(* Logix 5000 project; controller cal1615 1756-L62 rev 20.11; software revision 20.05; part 50 of 82 *)
(* tags used below, declared in another part *)
   FAULT : BOOL;   // Fault AFI
   metering_roll_alarm : TIMER;
   metering_roll_close : TIMER;
   p01_recipe_active : recipe;   // Active Recipe
   p01r02 : routine;   // System Misc Control
   p01r09_pb_global_reset : BOOL;   // System Modes PB: Global Fault Reset
   p02_dint_from_hmi : hmi_dint;
   p11r02_shutdown_temp : BOOL;   // Zone 1 Misc Control Safe Shutdown Temperature
   p11r30 : routine;   // Zone 1 Temperature Control
   p12r02_shutdown_temp : BOOL;   // Zone 2 Misc Control Safe Shutdown Temperature
   p12r30 : routine;   // Zone 2 Temperature Control
   p23_ai_ds_gap_dint : DINT;
   p23_ai_ds_masked_gap : REAL;
   p23_ai_lfl : REAL;   // Impreg Inputs LFL level
   p23_ai_metering_roll_amps : REAL;   // Impreg Analog Input Impreg Metering Roll Motor Current
   p23_ai_metering_roll_hz : REAL;   // Impreg Analog Input Impreg Metering Roll Motor Max Hz
   p23_ai_metering_roll_speed_fpm : REAL;   // Impreg Analog Input Impreg Roll Speed
   p23_ai_prs : REAL;   // Impreg Analog Inputs Impreg Enclosure Pressure
   p23_ai_servo_ds_position : REAL;   // Impreg Servo Drive Side Actual Position
   p23_ai_servo_ds_torque : REAL;   // Impreg Servo Drive Side Actual Torque
   p23_ai_servo_ds_velocity : REAL;   // Impreg Servo Drive Side Velocity Feedback
   p23_ai_servo_os_position : REAL;   // Impreg Inputs Servo Operator Side Position
   p23_ai_servo_os_velocity : REAL;   // Impreg Inputs Servo Operator Side Velocity
   p23_ai_supply_amps : REAL;   // Impreg Analog Inputs Supply Fan VFD Amps
   p23_ai_supply_hz : REAL;   // Impreg Analog Inputs Supply Fan VFD Hz
   p23_ai_supply_rpm : REAL;   // Impreg Analog Inputs Supply Fan RPM
   p23_ctr_gear_ratio : REAL;
   p23_ctr_lfl_input_max : REAL;
   p23_ctr_lfl_input_min : REAL;
   p23_ctr_lfl_output_max : REAL;
   p23_ctr_lfl_output_min : REAL;
   p23_ctr_roll_diameter_ft : REAL;
   p23_di_exhaust_speed_ok : BOOL;
   p23_di_filter_clean : BOOL;
   p23_di_impreg_exhaust_running : BOOL;
   p23_di_impreg_tank_up : BOOL;   // Input Impreg Dip Tank Up
   p23_di_metering_bar_close : BOOL;   // Impreg Input SSS: Metering Bar Close
   p23_di_metering_bar_open : BOOL;   // Impreg Input SSS: Metering Bar Open
   p23_di_metering_roll : acs800_di_normal;   // Impreg Digital Inputs Metering Roll VFD
   p23_di_servo_ds : servo_di;   // Impreg Digital Inputs Servo Drive Side
   p23_di_servo_os : servo_di;   // Impreg Digital Inputs Servo Operator Side
   p23_di_splice_jump : BOOL;   // Impreg Inputs PB: Splice Jump
   p23_di_spring : acs800_di_normal;
   p23_di_srv_ds_ok : BOOL;   // Impreg Inputs Metering Servo Drive Side Ok
   p23_di_srv_op_ok : BOOL;   // Impreg Inputs Metering Servo Operator Side Ok
   p23_di_supply : acs800_di_normal;   // Impreg Supply VFD VFD Inputs
   p23_di_supply_motor_therm : BOOL;   // Impreg Inputs Supply Fan Motor Thermostat
   p23_di_supply_speed_ok : BOOL;
   p23_di_tank_level_high : BOOL;   // Impreg Input Dip Impreg Level High
   p23_di_tank_level_low : BOOL;   // Impreg Input Dip Impreg Level Low
   p23_di_therm : BOOL;   // Impreg Inputs Metering Roll Motor Temperature Ok
   p23_di_though_level_low : BOOL;   // Impreg Input Dip Impreg Through Level Low
   p23_di_vfd_jog_fwd : BOOL;   // Impreg Input PB: VFD Jog FWD
   p23_di_vfd_jog_rev : BOOL;   // Impreg Input PB: VFD Jog REV
   p23_dint_to_hmi : DINT[17];   // Impreg Dint to HMI
   p23_do_enable_impreg_exhaust_fan : BOOL;   // Impreg Enclosure Digital Output Exhaust Fan Enable
   p23_do_impreg_nip_close : BOOL;   // Impreg Digital Output Impreg Nip close
   p23_param_lfl_hhl : REAL;   // Impreg Parameter LFL High High Limit
   p23_param_lfl_hl : REAL;   // Impreg Parameters LFL High Limit
   p23_param_servo_open_position : REAL;
   p23_param_zone_pressure : REAL;   // MOP HMI Iface Parameters Minimum Pressure
   p23r01 : routine;   // Impreg Main
   p23r02 : routine;   // Impreg Misc Control
   p23r02_fault_exists : BOOL;
   p23r02_open_pos_dint : DINT;
   p23r02_open_pos_real : REAL;
   p23r02_pb_start_exh : BOOL;
   p23r02_pb_stop_exh : BOOL;
   p23r02_request_nip_close : BOOL;   // Impreg Misc Control Request Nip Close
   p23r02_timer_fault : TIMER[4];   // Impreg Misc Control Timer Fault
   p23r02_timer_warning : TIMER[4];   // Impreg Misc Control Timer Warning
   p23r02_unack_fault : BOOL;   // Imperg Misc Control Unackn. Fault Exist
   p23r02_unack_warning : BOOL;   // Impreg Misc Control Unackn. Warning Exist
   p23r02_warning_exists : BOOL;
   p23r03 : routine;   // Impreg Inputs
   p23r03_hz : SYS_SCP;   // Impreg Roll Analog Inputs SCP Hz
   p23r03_impreg_lfl_monitor : SYS_SCP;   // Impreg Analog Inputs LFL Monitor Scaling
   p23r03_impreg_prs_input_max : REAL;
   p23r03_impreg_prs_input_min : REAL;
   p23r03_impreg_prs_output_max : REAL;
   p23r03_impreg_prs_output_min : REAL;
   p23r03_impreg_prs_scp : SYS_SCP;   // Impreg Analog Input Impreg Enclosure Pressure
   p23r03_metering_vfd_rpm_to_speed : SYS_RPM_TO_SPEED;   // Impreg Metering Roll Input VFD AI
   p23r04 : routine;   // Impreg Outputs
   p23r05 : routine;   // Impreg Dint to HMI
   p23r06 : routine;   // Impreg Real to HMI
   p23r07 : routine;   // Impreg Alarms
   p23r08 : routine;   // Impreg Warnings
   p23r09 : routine;   // Impreg Mode Selection
   p23r11 : routine;   // Impreg Servo Operator Side
   p23r12 : routine;   // Impreg Servo Drive Side
   p23r15 : routine;   // Impreg Metering Roll VFD
   p23r17_di_brake : BOOL;
   p23r17_di_therm : BOOL;

PROGRAM P23_Impreg   (* main routine R01_Main *)
VAR
   jog : BOOL;
   metering_roll : TIMER := (PRE := 4500);
   p23r17 : routine := (comment := -1073741714, fault := 48, fault_ack := 48);
   p23r17_request_line_run : BOOL;
END_VAR

ROUTINE R01_Main   (* ladder *)
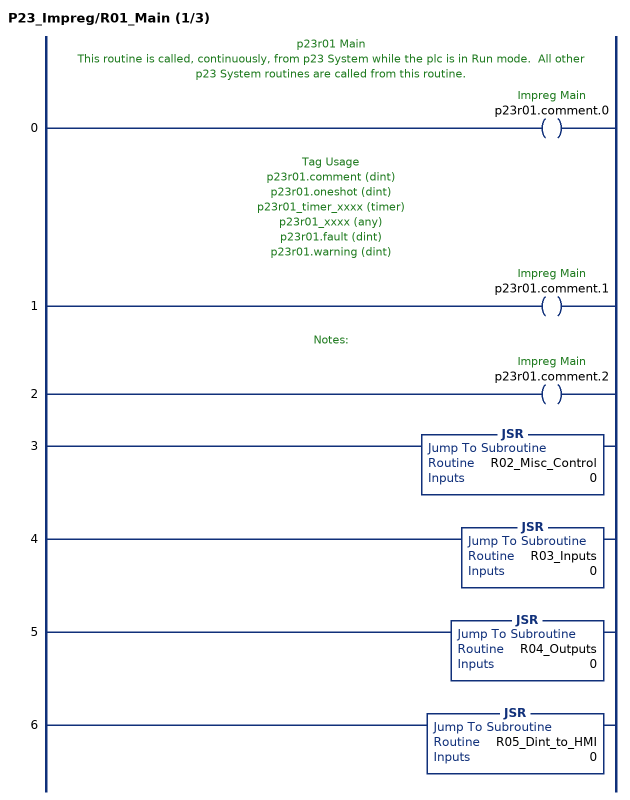
   // p23r01 Main
   // This routine is called, continuously, from p23 System while the plc is in Run mode.  All other p23 System routines are called from this routine.
   0: OTE(p23r01.comment.0);
   // Tag Usage
   // p23r01.comment (dint)
   // p23r01.oneshot (dint)
   // p23r01_timer_xxxx (timer)
   // p23r01_xxxx (any)
   // p23r01.fault (dint)
   // p23r01.warning (dint)
   1: OTE(p23r01.comment.1);
   // Notes:
   2: OTE(p23r01.comment.2);
   3: JSR(R02_Misc_Control,0);
   4: JSR(R03_Inputs,0);
   5: JSR(R04_Outputs,0);
   6: JSR(R05_Dint_to_HMI,0);
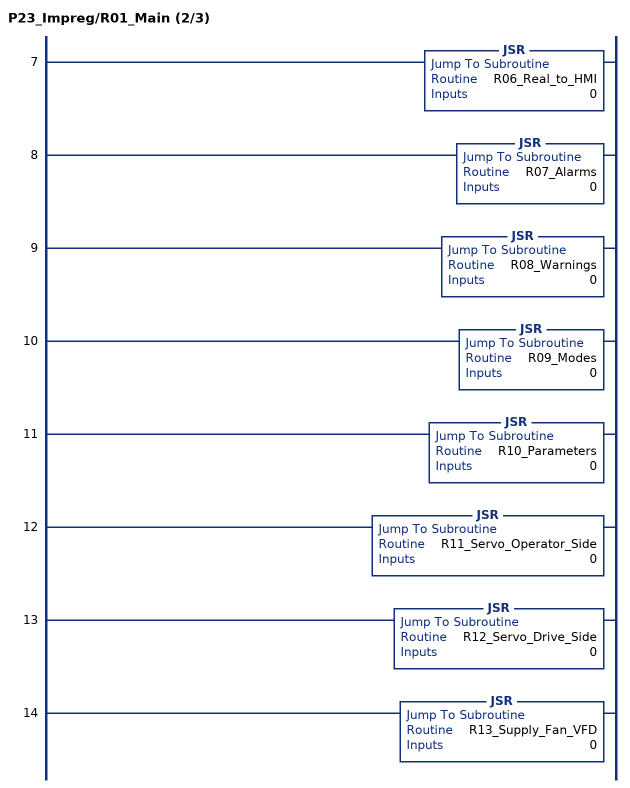
   7: JSR(R06_Real_to_HMI,0);
   8: JSR(R07_Alarms,0);
   9: JSR(R08_Warnings,0);
   10: JSR(R09_Modes,0);
   11: JSR(R10_Parameters,0);
   12: JSR(R11_Servo_Operator_Side,0);
   13: JSR(R12_Servo_Drive_Side,0);
   14: JSR(R13_Supply_Fan_VFD,0);
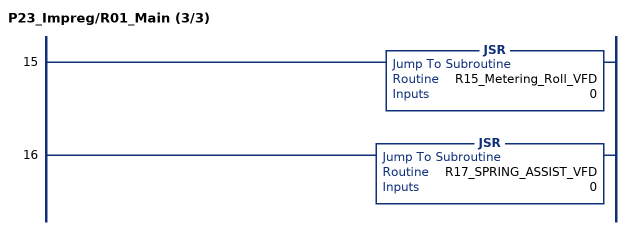
   15: JSR(R15_Metering_Roll_VFD,0);
   16: JSR(R17_SPRING_ASSIST_VFD,0);
END_ROUTINE

ROUTINE R02_Misc_Control   (* ladder *)
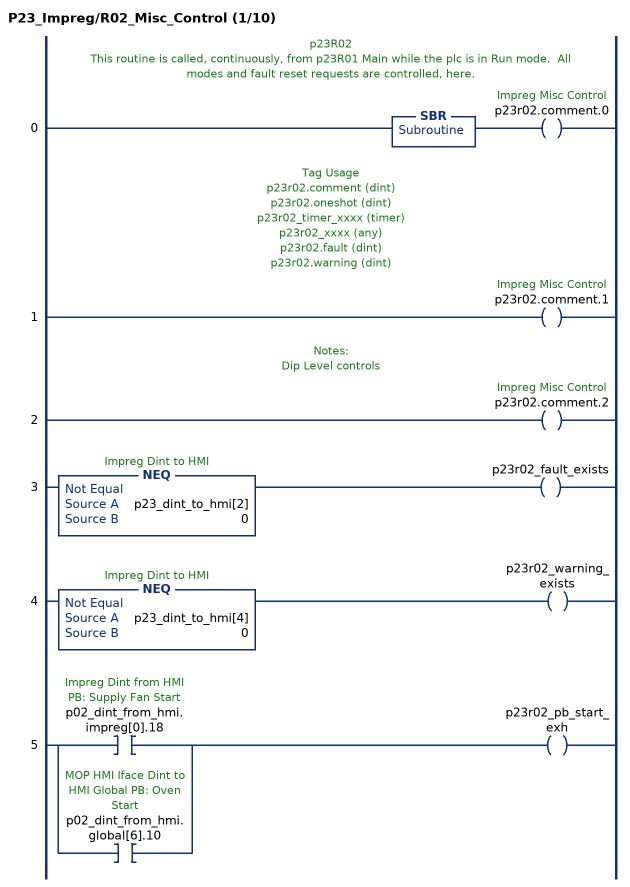
   // p23R02
   // This routine is called, continuously, from p23R01 Main while the plc is in Run mode.  All modes and fault reset requests are controlled, here.
   0: SBR()OTE(p23r02.comment.0);
   // Tag Usage
   // p23r02.comment (dint)
   // p23r02.oneshot (dint)
   // p23r02_timer_xxxx (timer)
   // p23r02_xxxx (any)
   // p23r02.fault (dint)
   // p23r02.warning (dint)
   1: OTE(p23r02.comment.1);
   // Notes:
   // Dip Level controls
   2: OTE(p23r02.comment.2);
   3: NEQ(p23_dint_to_hmi[2],0)OTE(p23r02_fault_exists);
   4: NEQ(p23_dint_to_hmi[4],0)OTE(p23r02_warning_exists);
   5: [XIC(p02_dint_from_hmi.impreg[0].18) ,XIC(p02_dint_from_hmi.global[6].10) ]OTE(p23r02_pb_start_exh);
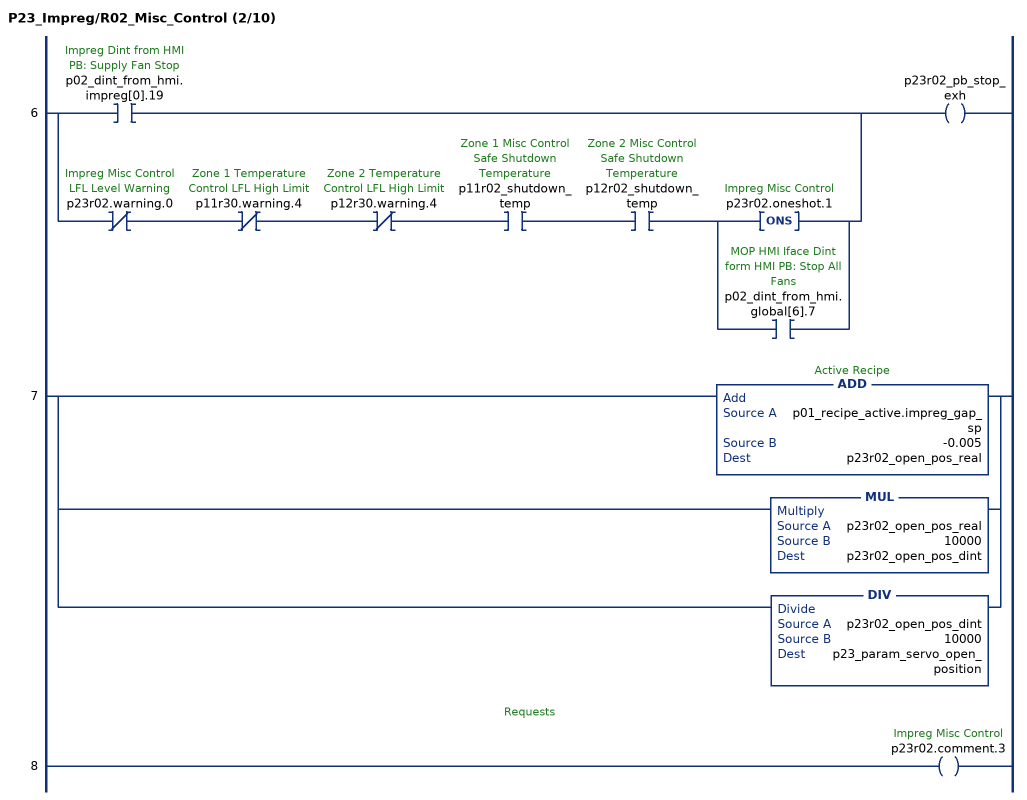
   6: [XIC(p02_dint_from_hmi.impreg[0].19) ,XIO(p23r02.warning.0) XIO(p11r30.warning.4) XIO(p12r30.warning.4) XIC(p11r02_shutdown_temp) XIC(p12r02_shutdown_temp) [ONS(p23r02.oneshot.1) ,XIC(p02_dint_from_hmi.global[6].7) ] ]OTE(p23r02_pb_stop_exh);
   7: [ADD(p01_recipe_active.impreg_gap_sp,-0.005,p23r02_open_pos_real) ,MUL(p23r02_open_pos_real,10000,p23r02_open_pos_dint) ,DIV(p23r02_open_pos_dint,10000,p23_param_servo_open_position) ];
   // Requests
   8: OTE(p23r02.comment.3);
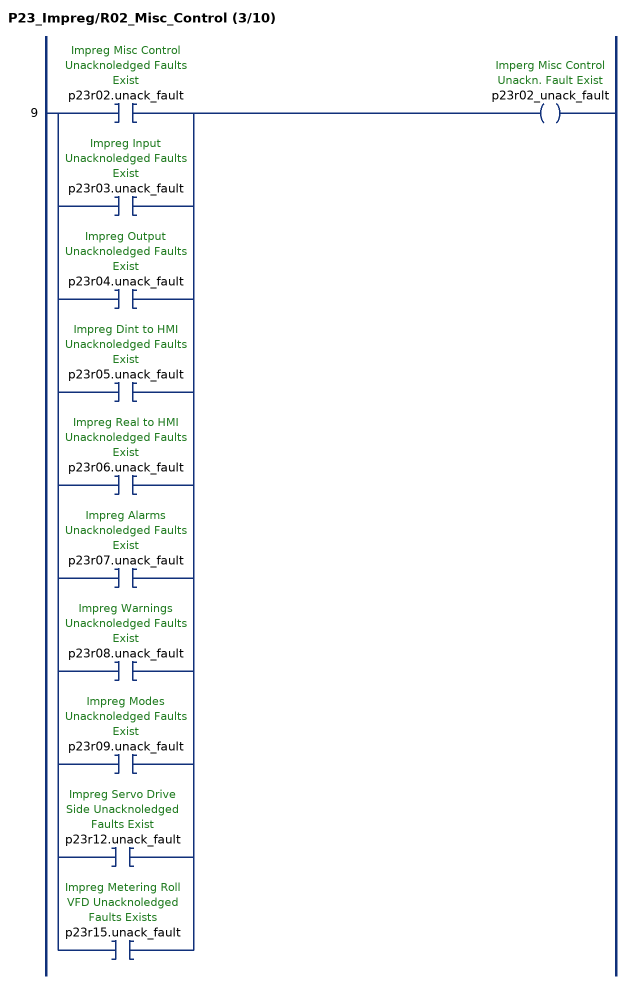
   9: [XIC(p23r02.unack_fault) ,XIC(p23r03.unack_fault) ,XIC(p23r04.unack_fault) ,XIC(p23r05.unack_fault) ,XIC(p23r06.unack_fault) ,XIC(p23r07.unack_fault) ,XIC(p23r08.unack_fault) ,XIC(p23r09.unack_fault) ,XIC(p23r12.unack_fault) ,XIC(p23r15.unack_fault) ]OTE(p23r02_unack_fault);
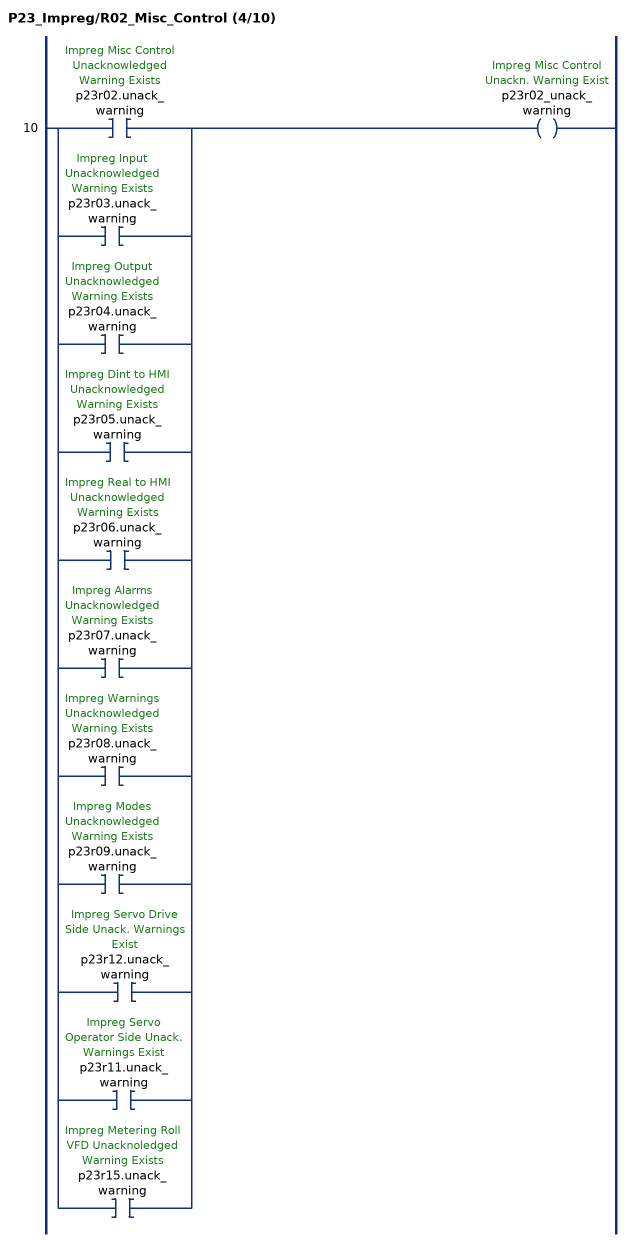
   10: [XIC(p23r02.unack_warning) ,XIC(p23r03.unack_warning) ,XIC(p23r04.unack_warning) ,XIC(p23r05.unack_warning) ,XIC(p23r06.unack_warning) ,XIC(p23r07.unack_warning) ,XIC(p23r08.unack_warning) ,XIC(p23r09.unack_warning) ,XIC(p23r12.unack_warning) ,XIC(p23r11.unack_warning) ,XIC(p23r15.unack_warning) ]OTE(p23r02_unack_warning);
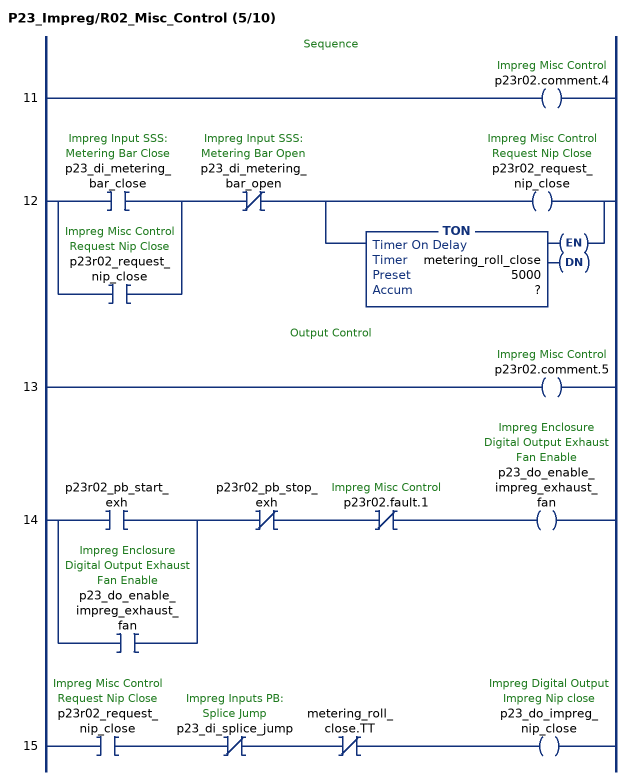
   // Sequence
   11: OTE(p23r02.comment.4);
   12: [XIC(p23_di_metering_bar_close) ,XIC(p23r02_request_nip_close) ]XIO(p23_di_metering_bar_open)[OTE(p23r02_request_nip_close) ,TON(metering_roll_close,?,?) ];
   // Output Control
   13: OTE(p23r02.comment.5);
   14: [XIC(p23r02_pb_start_exh) ,XIC(p23_do_enable_impreg_exhaust_fan) ]XIO(p23r02_pb_stop_exh)XIO(p23r02.fault.1)OTE(p23_do_enable_impreg_exhaust_fan);
   15: XIC(p23r02_request_nip_close)XIO(p23_di_splice_jump)XIO(metering_roll_close.TT)OTE(p23_do_impreg_nip_close);
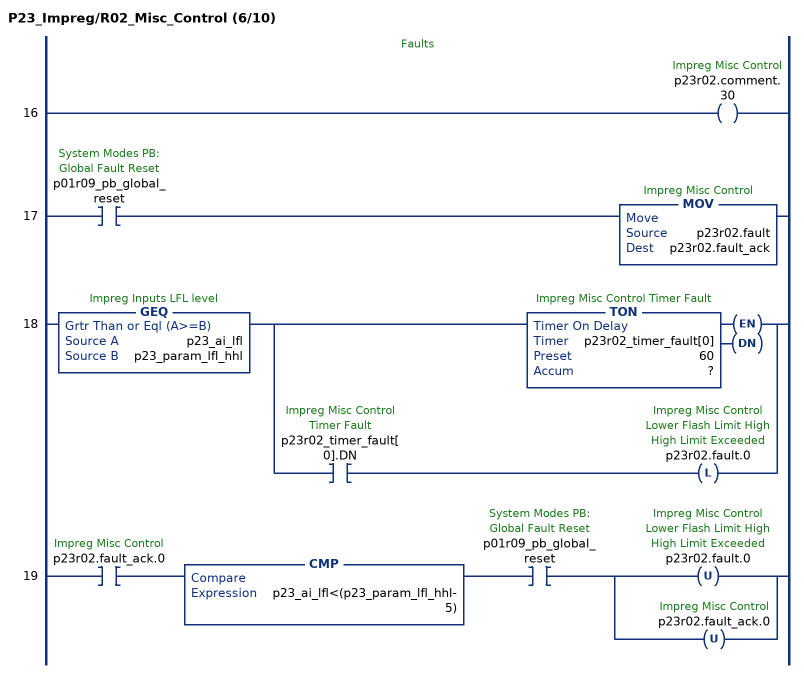
   // Faults
   16: OTE(p23r02.comment.30);
   17: XIC(p01r09_pb_global_reset)MOV(p23r02.fault,p23r02.fault_ack);
   18: GEQ(p23_ai_lfl,p23_param_lfl_hhl)[TON(p23r02_timer_fault[0],?,?) ,XIC(p23r02_timer_fault[0].DN) OTL(p23r02.fault.0) ];
   19: XIC(p23r02.fault_ack.0)CMP(p23_ai_lfl<(p23_param_lfl_hhl-5))XIC(p01r09_pb_global_reset)[OTU(p23r02.fault.0) ,OTU(p23r02.fault_ack.0) ];
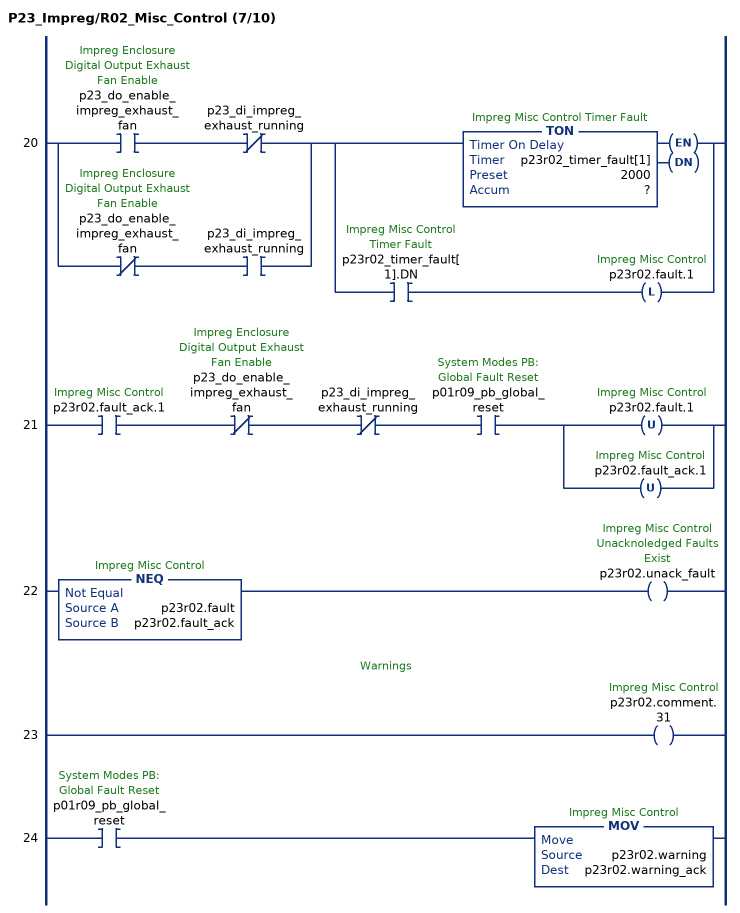
   20: [XIC(p23_do_enable_impreg_exhaust_fan) XIO(p23_di_impreg_exhaust_running) ,XIO(p23_do_enable_impreg_exhaust_fan) XIC(p23_di_impreg_exhaust_running) ][TON(p23r02_timer_fault[1],?,?) ,XIC(p23r02_timer_fault[1].DN) OTL(p23r02.fault.1) ];
   21: XIC(p23r02.fault_ack.1)XIO(p23_do_enable_impreg_exhaust_fan)XIO(p23_di_impreg_exhaust_running)XIC(p01r09_pb_global_reset)[OTU(p23r02.fault.1) ,OTU(p23r02.fault_ack.1) ];
   22: NEQ(p23r02.fault,p23r02.fault_ack)OTE(p23r02.unack_fault);
   // Warnings
   23: OTE(p23r02.comment.31);
   24: XIC(p01r09_pb_global_reset)MOV(p23r02.warning,p23r02.warning_ack);
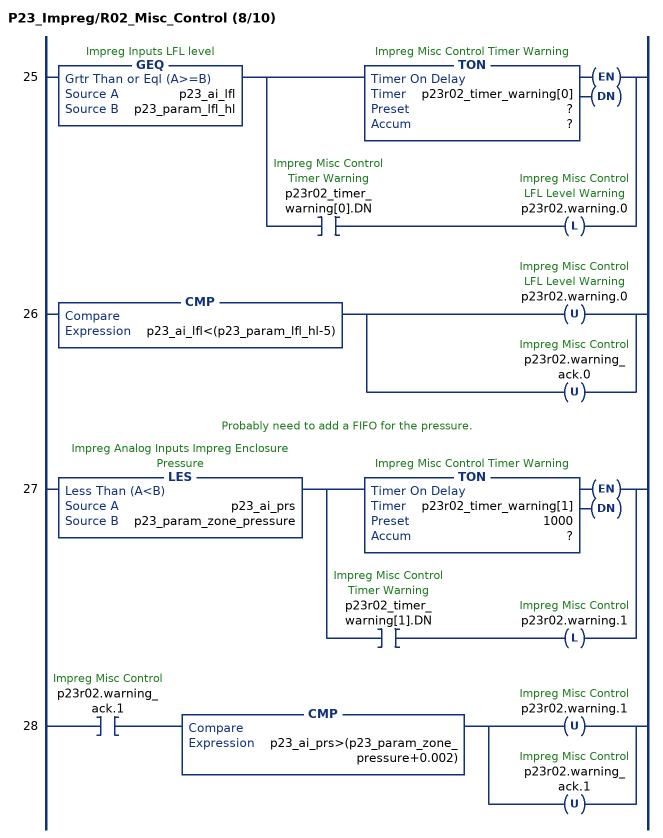
   25: GEQ(p23_ai_lfl,p23_param_lfl_hl)[TON(p23r02_timer_warning[0],?,?) ,XIC(p23r02_timer_warning[0].DN) OTL(p23r02.warning.0) ];
   26: CMP(p23_ai_lfl<(p23_param_lfl_hl-5))[OTU(p23r02.warning.0) ,OTU(p23r02.warning_ack.0) ];
   // Probably need to add a FIFO for the pressure.
   27: LES(p23_ai_prs,p23_param_zone_pressure)[TON(p23r02_timer_warning[1],?,?) ,XIC(p23r02_timer_warning[1].DN) OTL(p23r02.warning.1) ];
   28: XIC(p23r02.warning_ack.1)CMP(p23_ai_prs>(p23_param_zone_pressure+0.002))[OTU(p23r02.warning.1) ,OTU(p23r02.warning_ack.1) ];
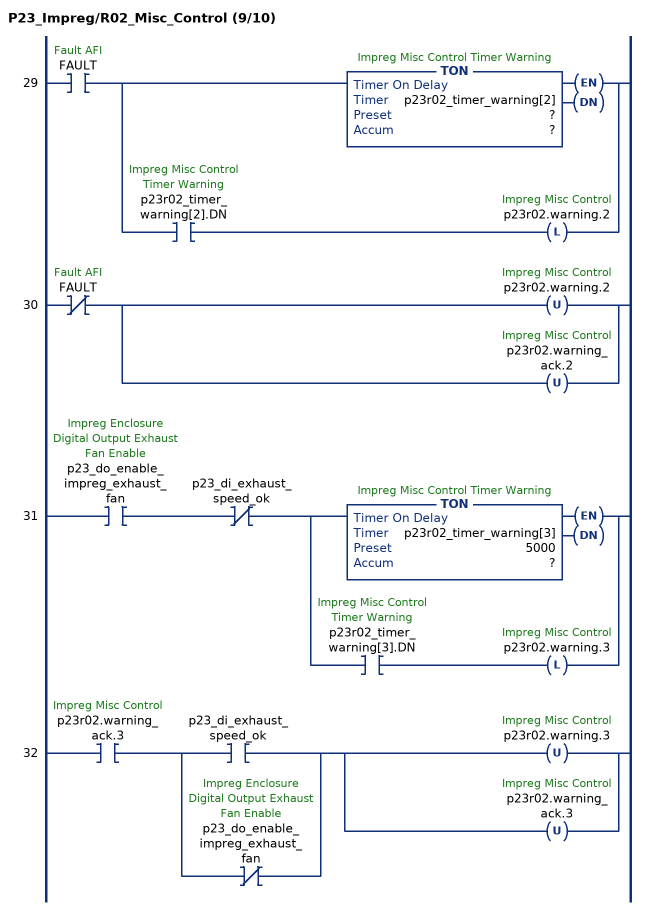
   29: XIC(FAULT)[TON(p23r02_timer_warning[2],?,?) ,XIC(p23r02_timer_warning[2].DN) OTL(p23r02.warning.2) ];
   30: XIO(FAULT)[OTU(p23r02.warning.2) ,OTU(p23r02.warning_ack.2) ];
   31: XIC(p23_do_enable_impreg_exhaust_fan)XIO(p23_di_exhaust_speed_ok)[TON(p23r02_timer_warning[3],?,?) ,XIC(p23r02_timer_warning[3].DN) OTL(p23r02.warning.3) ];
   32: XIC(p23r02.warning_ack.3)[XIC(p23_di_exhaust_speed_ok) ,XIO(p23_do_enable_impreg_exhaust_fan) ][OTU(p23r02.warning.3) ,OTU(p23r02.warning_ack.3) ];
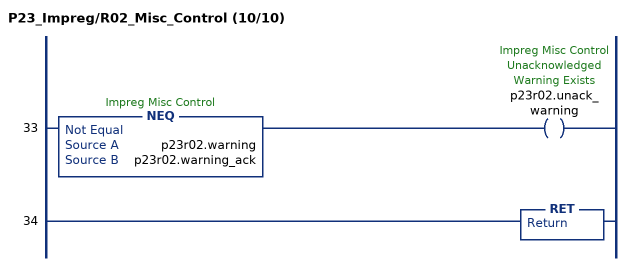
   33: NEQ(p23r02.warning,p23r02.warning_ack)OTE(p23r02.unack_warning);
   34: RET();
END_ROUTINE

ROUTINE R03_Inputs   (* ladder *)
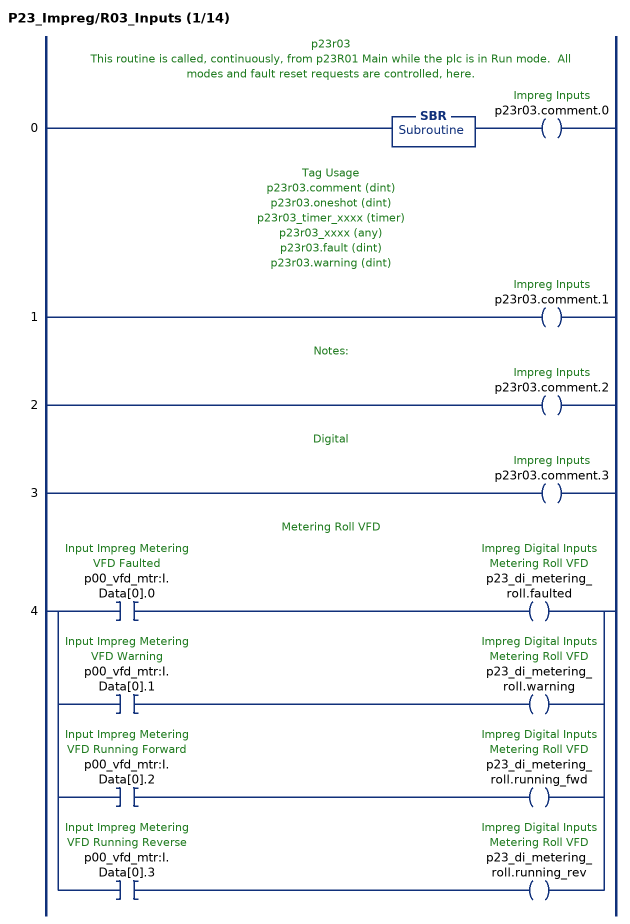
   // p23r03
   // This routine is called, continuously, from p23R01 Main while the plc is in Run mode.  All modes and fault reset requests are controlled, here.
   0: SBR()OTE(p23r03.comment.0);
   // Tag Usage
   // p23r03.comment (dint)
   // p23r03.oneshot (dint)
   // p23r03_timer_xxxx (timer)
   // p23r03_xxxx (any)
   // p23r03.fault (dint)
   // p23r03.warning (dint)
   1: OTE(p23r03.comment.1);
   // Notes:
   2: OTE(p23r03.comment.2);
   // Digital
   3: OTE(p23r03.comment.3);
   // Metering Roll VFD
   4: [XIC(p00_vfd_mtr:I.Data[0].0) OTE(p23_di_metering_roll.faulted) ,XIC(p00_vfd_mtr:I.Data[0].1) OTE(p23_di_metering_roll.warning) ,XIC(p00_vfd_mtr:I.Data[0].2) OTE(p23_di_metering_roll.running_fwd) ,XIC(p00_vfd_mtr:I.Data[0].3) OTE(p23_di_metering_roll.running_rev) ];
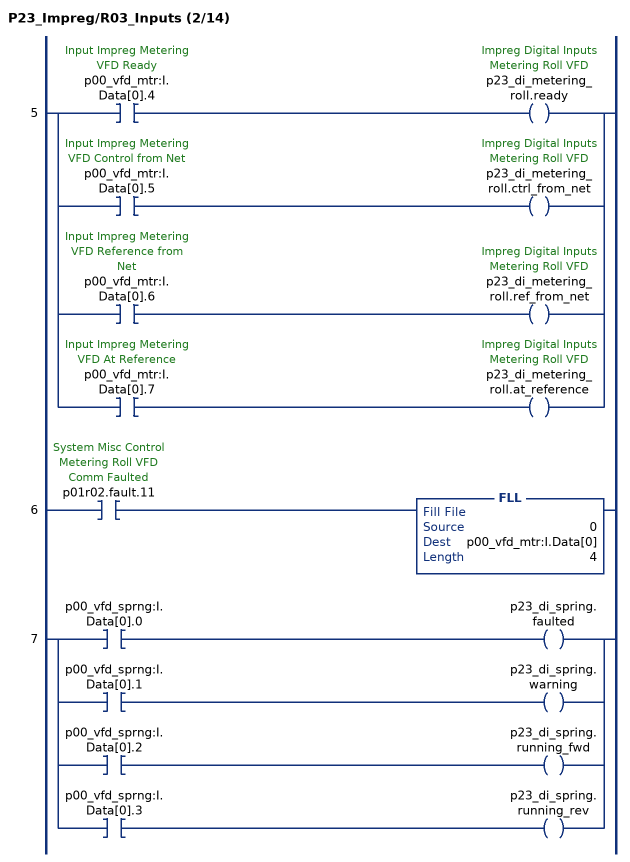
   5: [XIC(p00_vfd_mtr:I.Data[0].4) OTE(p23_di_metering_roll.ready) ,XIC(p00_vfd_mtr:I.Data[0].5) OTE(p23_di_metering_roll.ctrl_from_net) ,XIC(p00_vfd_mtr:I.Data[0].6) OTE(p23_di_metering_roll.ref_from_net) ,XIC(p00_vfd_mtr:I.Data[0].7) OTE(p23_di_metering_roll.at_reference) ];
   6: XIC(p01r02.fault.11)FLL(0,p00_vfd_mtr:I.Data[0],4);
   7: [XIC(p00_vfd_sprng:I.Data[0].0) OTE(p23_di_spring.faulted) ,XIC(p00_vfd_sprng:I.Data[0].1) OTE(p23_di_spring.warning) ,XIC(p00_vfd_sprng:I.Data[0].2) OTE(p23_di_spring.running_fwd) ,XIC(p00_vfd_sprng:I.Data[0].3) OTE(p23_di_spring.running_rev) ];
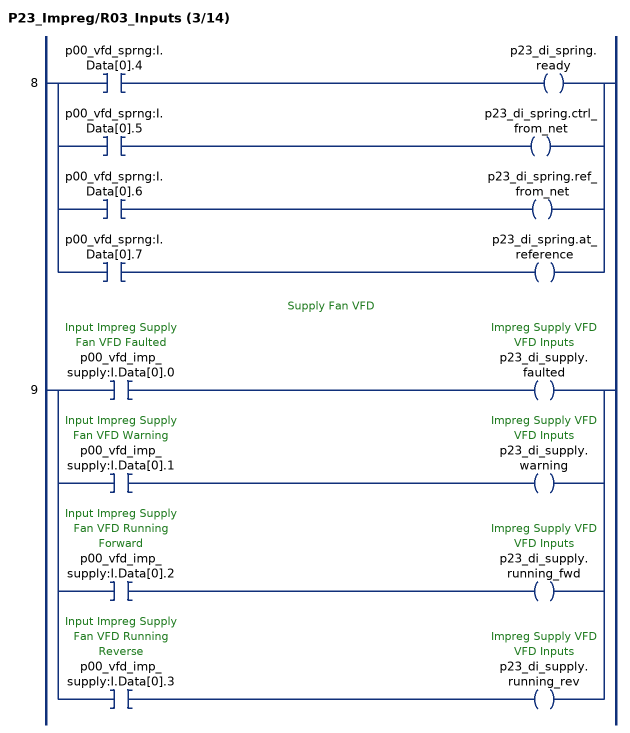
   8: [XIC(p00_vfd_sprng:I.Data[0].4) OTE(p23_di_spring.ready) ,XIC(p00_vfd_sprng:I.Data[0].5) OTE(p23_di_spring.ctrl_from_net) ,XIC(p00_vfd_sprng:I.Data[0].6) OTE(p23_di_spring.ref_from_net) ,XIC(p00_vfd_sprng:I.Data[0].7) OTE(p23_di_spring.at_reference) ];
   // Supply Fan VFD
   9: [XIC(p00_vfd_imp_supply:I.Data[0].0) OTE(p23_di_supply.faulted) ,XIC(p00_vfd_imp_supply:I.Data[0].1) OTE(p23_di_supply.warning) ,XIC(p00_vfd_imp_supply:I.Data[0].2) OTE(p23_di_supply.running_fwd) ,XIC(p00_vfd_imp_supply:I.Data[0].3) OTE(p23_di_supply.running_rev) ];
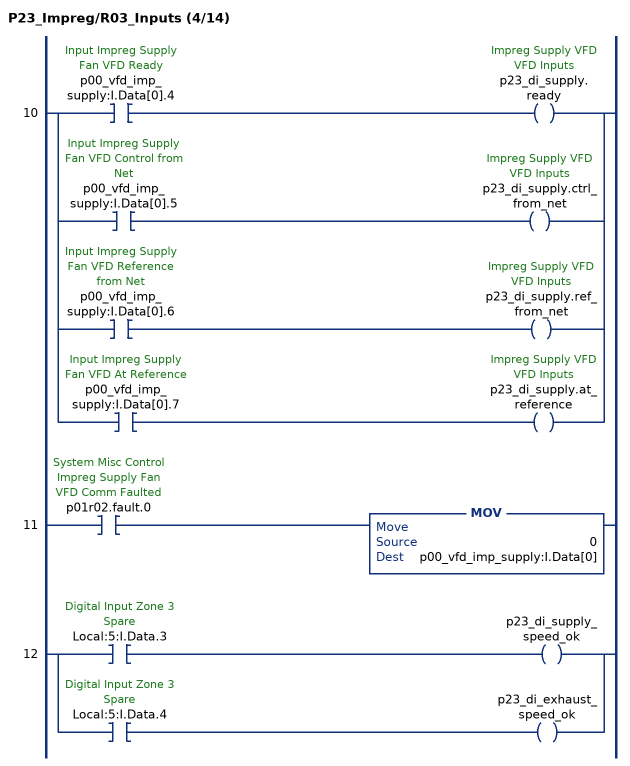
   10: [XIC(p00_vfd_imp_supply:I.Data[0].4) OTE(p23_di_supply.ready) ,XIC(p00_vfd_imp_supply:I.Data[0].5) OTE(p23_di_supply.ctrl_from_net) ,XIC(p00_vfd_imp_supply:I.Data[0].6) OTE(p23_di_supply.ref_from_net) ,XIC(p00_vfd_imp_supply:I.Data[0].7) OTE(p23_di_supply.at_reference) ];
   11: XIC(p01r02.fault.0)MOV(0,p00_vfd_imp_supply:I.Data[0]);
   12: [XIC(Local:5:I.Data.3) OTE(p23_di_supply_speed_ok) ,XIC(Local:5:I.Data.4) OTE(p23_di_exhaust_speed_ok) ];
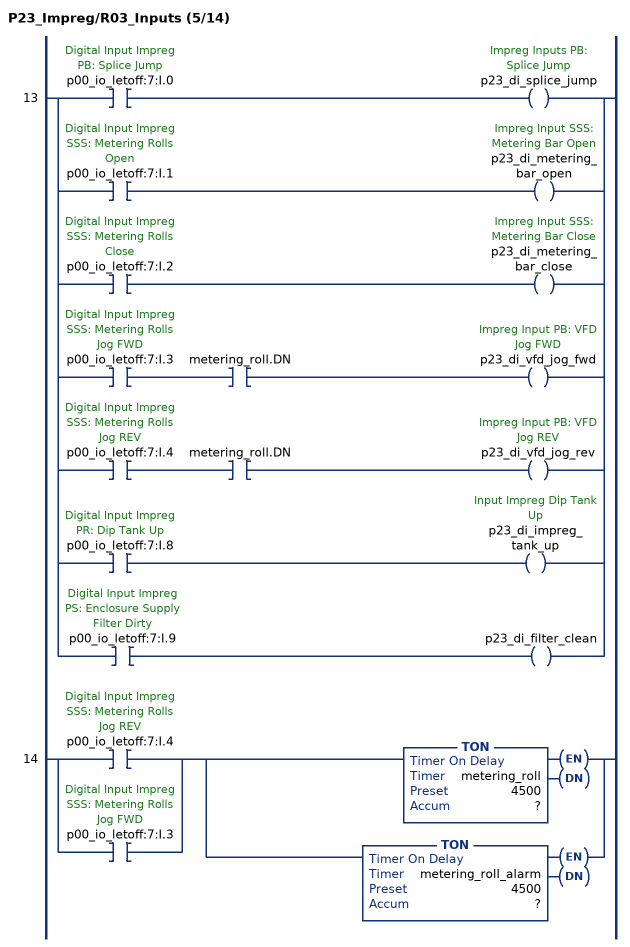
   13: [XIC(p00_io_letoff:7:I.0) OTE(p23_di_splice_jump) ,XIC(p00_io_letoff:7:I.1) OTE(p23_di_metering_bar_open) ,XIC(p00_io_letoff:7:I.2) OTE(p23_di_metering_bar_close) ,XIC(p00_io_letoff:7:I.3) XIC(metering_roll.DN) OTE(p23_di_vfd_jog_fwd) ,XIC(p00_io_letoff:7:I.4) XIC(metering_roll.DN) OTE(p23_di_vfd_jog_rev) ,XIC(p00_io_letoff:7:I.8) OTE(p23_di_impreg_tank_up) ,XIC(p00_io_letoff:7:I.9) OTE(p23_di_filter_clean) ];
   14: [XIC(p00_io_letoff:7:I.4) ,XIC(p00_io_letoff:7:I.3) ][TON(metering_roll,?,?) ,TON(metering_roll_alarm,?,?) ];
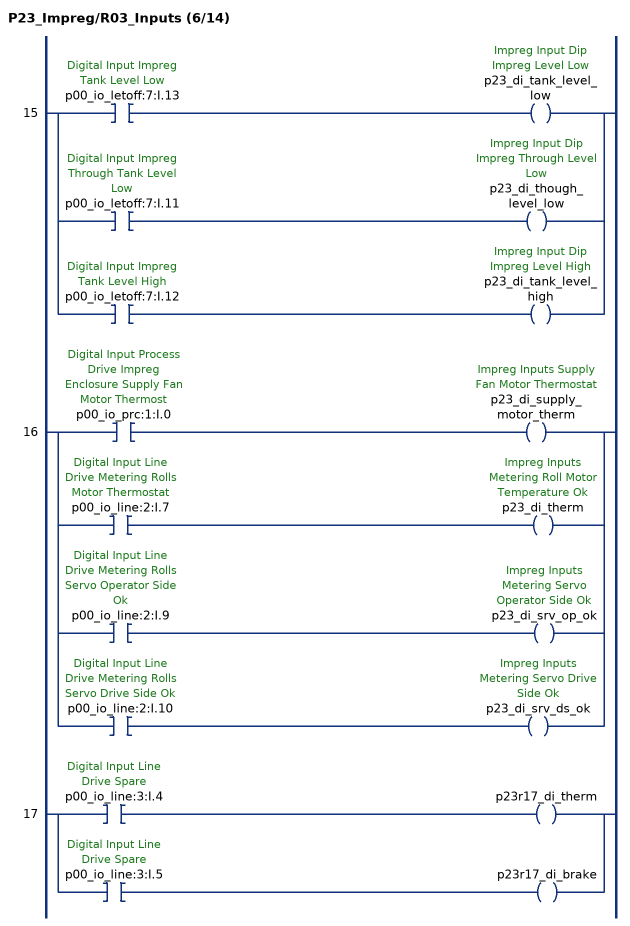
   15: [XIC(p00_io_letoff:7:I.13) OTE(p23_di_tank_level_low) ,XIC(p00_io_letoff:7:I.11) OTE(p23_di_though_level_low) ,XIC(p00_io_letoff:7:I.12) OTE(p23_di_tank_level_high) ];
   16: [XIC(p00_io_prc:1:I.0) OTE(p23_di_supply_motor_therm) ,XIC(p00_io_line:2:I.7) OTE(p23_di_therm) ,XIC(p00_io_line:2:I.9) OTE(p23_di_srv_op_ok) ,XIC(p00_io_line:2:I.10) OTE(p23_di_srv_ds_ok) ];
   17: [XIC(p00_io_line:3:I.4) OTE(p23r17_di_therm) ,XIC(p00_io_line:3:I.5) OTE(p23r17_di_brake) ];
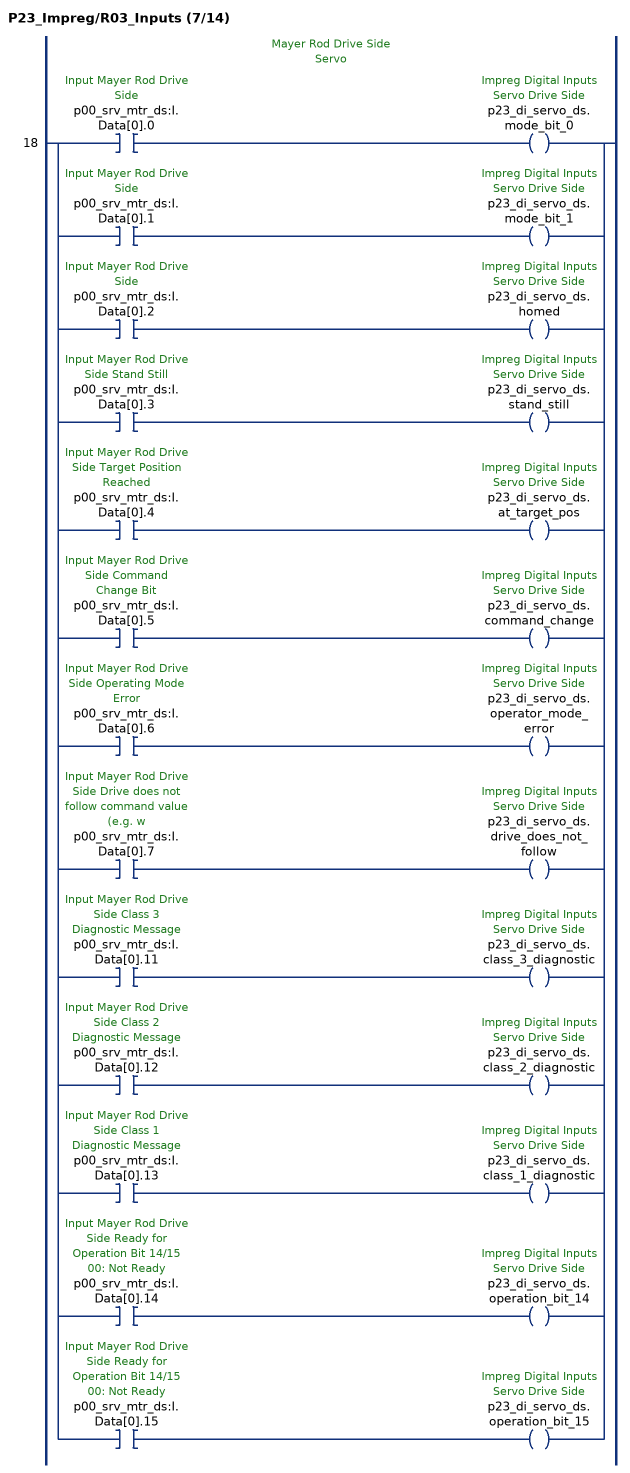
   // Mayer Rod Drive Side
   // Servo
   18: [XIC(p00_srv_mtr_ds:I.Data[0].0) OTE(p23_di_servo_ds.mode_bit_0) ,XIC(p00_srv_mtr_ds:I.Data[0].1) OTE(p23_di_servo_ds.mode_bit_1) ,XIC(p00_srv_mtr_ds:I.Data[0].2) OTE(p23_di_servo_ds.homed) ,XIC(p00_srv_mtr_ds:I.Data[0].3) OTE(p23_di_servo_ds.stand_still) ,XIC(p00_srv_mtr_ds:I.Data[0].4) OTE(p23_di_servo_ds.at_target_pos) ,XIC(p00_srv_mtr_ds:I.Data[0].5) OTE(p23_di_servo_ds.command_change) ,XIC(p00_srv_mtr_ds:I.Data[0].6) OTE(p23_di_servo_ds.operator_mode_error) ,XIC(p00_srv_mtr_ds:I.Data[0].7) OTE(p23_di_servo_ds.drive_does_not_follow) ,XIC(p00_srv_mtr_ds:I.Data[0].11) OTE(p23_di_servo_ds.class_3_diagnostic) ,XIC(p00_srv_mtr_ds:I.Data[0].12) OTE(p23_di_servo_ds.class_2_diagnostic) ,XIC(p00_srv_mtr_ds:I.Data[0].13) OTE(p23_di_servo_ds.class_1_diagnostic) ,XIC(p00_srv_mtr_ds:I.Data[0].14) OTE(p23_di_servo_ds.operation_bit_14) ,XIC(p00_srv_mtr_ds:I.Data[0].15) OTE(p23_di_servo_ds.operation_bit_15) ];
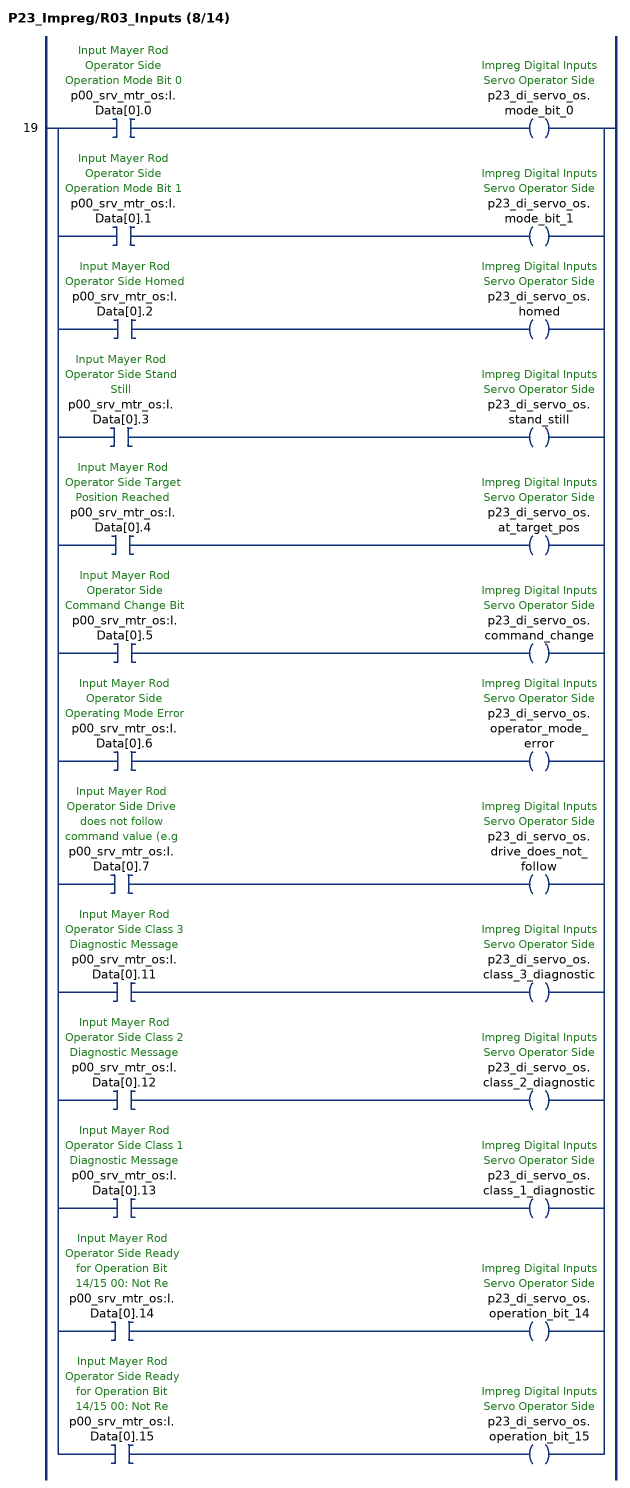
   19: [XIC(p00_srv_mtr_os:I.Data[0].0) OTE(p23_di_servo_os.mode_bit_0) ,XIC(p00_srv_mtr_os:I.Data[0].1) OTE(p23_di_servo_os.mode_bit_1) ,XIC(p00_srv_mtr_os:I.Data[0].2) OTE(p23_di_servo_os.homed) ,XIC(p00_srv_mtr_os:I.Data[0].3) OTE(p23_di_servo_os.stand_still) ,XIC(p00_srv_mtr_os:I.Data[0].4) OTE(p23_di_servo_os.at_target_pos) ,XIC(p00_srv_mtr_os:I.Data[0].5) OTE(p23_di_servo_os.command_change) ,XIC(p00_srv_mtr_os:I.Data[0].6) OTE(p23_di_servo_os.operator_mode_error) ,XIC(p00_srv_mtr_os:I.Data[0].7) OTE(p23_di_servo_os.drive_does_not_follow) ,XIC(p00_srv_mtr_os:I.Data[0].11) OTE(p23_di_servo_os.class_3_diagnostic) ,XIC(p00_srv_mtr_os:I.Data[0].12) OTE(p23_di_servo_os.class_2_diagnostic) ,XIC(p00_srv_mtr_os:I.Data[0].13) OTE(p23_di_servo_os.class_1_diagnostic) ,XIC(p00_srv_mtr_os:I.Data[0].14) OTE(p23_di_servo_os.operation_bit_14) ,XIC(p00_srv_mtr_os:I.Data[0].15) OTE(p23_di_servo_os.operation_bit_15) ];
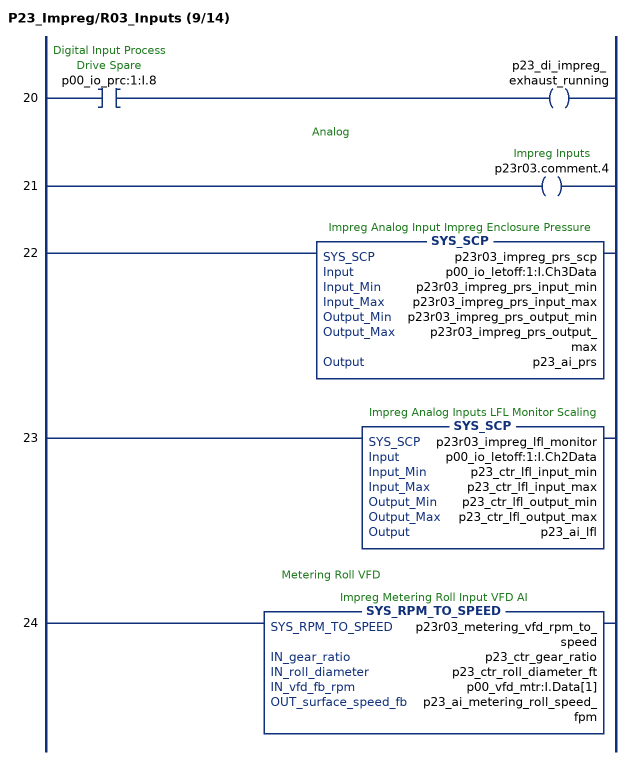
   20: XIC(p00_io_prc:1:I.8)OTE(p23_di_impreg_exhaust_running);
   // Analog
   21: OTE(p23r03.comment.4);
   22: SYS_SCP(p23r03_impreg_prs_scp,p00_io_letoff:1:I.Ch3Data,p23r03_impreg_prs_input_min,p23r03_impreg_prs_input_max,p23r03_impreg_prs_output_min,p23r03_impreg_prs_output_max,p23_ai_prs);
   23: SYS_SCP(p23r03_impreg_lfl_monitor,p00_io_letoff:1:I.Ch2Data,p23_ctr_lfl_input_min,p23_ctr_lfl_input_max,p23_ctr_lfl_output_min,p23_ctr_lfl_output_max,p23_ai_lfl);
   // Metering Roll VFD
   24: SYS_RPM_TO_SPEED(p23r03_metering_vfd_rpm_to_speed,p23_ctr_gear_ratio,p23_ctr_roll_diameter_ft,p00_vfd_mtr:I.Data[1],p23_ai_metering_roll_speed_fpm);
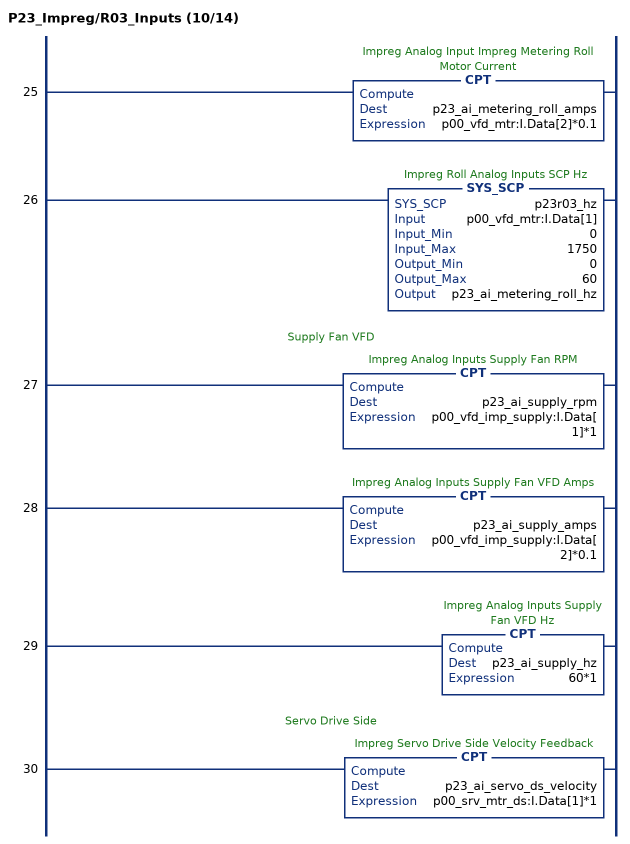
   25: CPT(p23_ai_metering_roll_amps,p00_vfd_mtr:I.Data[2]*0.1);
   26: SYS_SCP(p23r03_hz,p00_vfd_mtr:I.Data[1],0,1750,0,60,p23_ai_metering_roll_hz);
   // Supply Fan VFD
   27: CPT(p23_ai_supply_rpm,p00_vfd_imp_supply:I.Data[1]*1);
   28: CPT(p23_ai_supply_amps,p00_vfd_imp_supply:I.Data[2]*0.1);
   29: CPT(p23_ai_supply_hz,60*1);
   // Servo Drive Side
   30: CPT(p23_ai_servo_ds_velocity,p00_srv_mtr_ds:I.Data[1]*1);
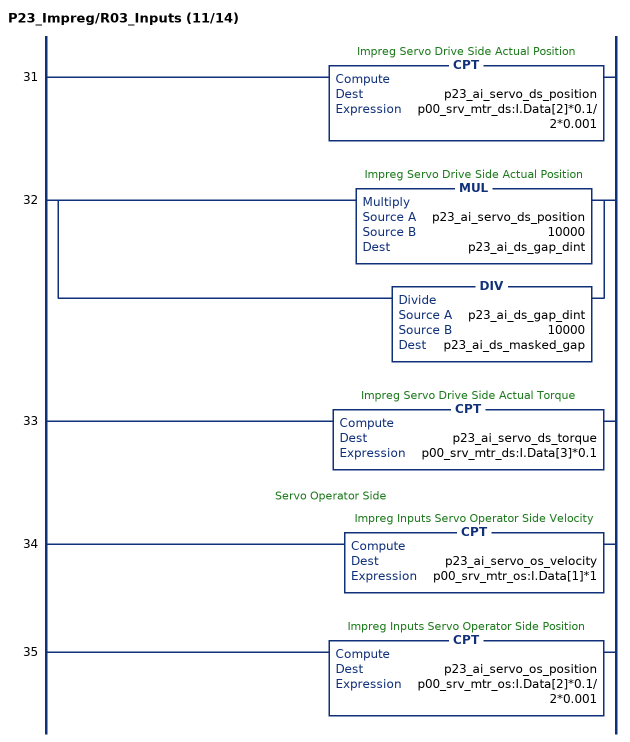
   31: CPT(p23_ai_servo_ds_position,p00_srv_mtr_ds:I.Data[2]*0.1/2*0.001);
   32: [MUL(p23_ai_servo_ds_position,10000,p23_ai_ds_gap_dint) ,DIV(p23_ai_ds_gap_dint,10000,p23_ai_ds_masked_gap) ];
   33: CPT(p23_ai_servo_ds_torque,p00_srv_mtr_ds:I.Data[3]*0.1);
   // Servo Operator Side
   34: CPT(p23_ai_servo_os_velocity,p00_srv_mtr_os:I.Data[1]*1);
   35: CPT(p23_ai_servo_os_position,p00_srv_mtr_os:I.Data[2]*0.1/2*0.001);
